// TIA Portal V19 export
DATA_BLOCK "SetpointsV0101Condensate"   // DB114
{ S7_Optimized_Access := 'TRUE' }
// stored: AutoNumber false, MemoryReserve 0
   VAR RETAIN
      TT0178_CondenseHigh : Real := 100.0;   // TT0178 Condensate Temperature Fault High
      TT0178_CondenseLow : Real := 50.0;   // TT0178 Condensate Temperature Fault Low
      TT0930_Low_Prod : Real := 100.0;   // TT0930 Low Temperature
      TT0930_Low_SIP : Real := 100.0;   // TT0930 Low Temperature
      TT0931_Low_Prod : Real := 100.0;   // TT0930 Low Temperature
      CT0930_High : Real := 100.0;   // CT0930 High Conductivity - Suspect product in Condensate
   END_VAR
BEGIN
END_DATA_BLOCK
